(* IEC 61131-3 sources: repolevel_ST_code_completion/output/0122完整版本_无planner目前sota/repoeval_Proxy_Application/readful_result, 2 files *)

(* ---- Proxy.st ---- *)
{attribute 'enable_dynamic_creation'}
FUNCTION_BLOCK Proxy IMPLEMENTS Subject_Interface
VAR
refToRealSubject : POINTER TO Realsubject; // Declare refToRealSubject uniquely
iTempPassword : INT; // Declare iTempPassword uniquely
iRealPassword : INT := 1234; // Declare all instance variables globally
END_VAR

METHOD fb_init
VAR_INPUT
bInitRetains : BOOL; // Input Variables
bInCopyCode : BOOL;
ptrToRealSubject : POINTER TO Realsubject;
iSetValue : INT;
bReadWrite : BOOL;
END_VAR

// Correct logic for initialization
IF ptrToRealSubject <> 0 THEN
refToRealSubject := ptrToRealSubject; // Correct assignment between pointers
END_IF;

IF bReadWrite THEN
IF iTempPassword = iRealPassword THEN
 refToRealSubject^.iProp := iSetValue; // Modify external property
END_IF;
ELSE
IF iTempPassword = iRealPassword THEN
 RETURN; // Read-only mode, return successful test but no data
ELSE
 RETURN; // Invalid password, no operation performed
END_IF;
END_IF;
END_METHOD;

END_FUNCTION_BLOCK

(* ---- Realsubject.st ---- *)
{attribute 'enable_dynamic_creation'}
FUNCTION_BLOCK Realsubject IMPLEMENTS  Subject_Interface
VAR_INPUT
END_VAR
VAR_OUTPUT
END_VAR
VAR
    // Variable to get and set values
    iProp: INT;
END_VAR

VAR_STAT
END_VAR

METHOD Get_Method : INT
RETURN iProp; // Correct return of iProp value
END_METHOD

METHOD Set_Method
iProp := iProp; // Assume intent is copying within itself. No `num` variable defined.
END_METHOD
END_FUNCTION_BLOCK
